// TIA Portal project "S7-1500 için Kod Çözücü(DECO) Komutu" (V18)

(* hardware
DEVICE "S7-1500/ET200MP station_1"  S7-1500 station
   slot 0: "Rail_0"  Rack  6ES7 590-1***0-0AA0
   slot 1: "PLC_1"  CPU 1512C-1 PN  6ES7 512-1CK00-0AB0  V2.8
      slot 3: "CPU display_1"  6ES7591-1AA00-0AA0
      slot 32768: "PROFINET interface_1"  X1
         slot 32769: "Port_1"  X1 P1
         slot 32770: "Port_2"  X1 P2
      slot 34817: "Virtual CP interface port_1"  Virtual CP interface port  Virtual CP interface port
*)

// ===== PLC "PLC_1"  CPU 1512C-1 PN =====

VAR_GLOBAL   // PLC tag table "Default tag table"
   "Tag_1" AT %I0.0 : Bool;
   "Tag_2" AT %MW10 : Int;
   "Tag_3" AT %Q0.0 : Bool;
   "Tag_4" AT %I0.1 : Bool;
   "Tag_5" AT %Q0.1 : Bool;
   "Tag_6" AT %MW11 : Int;
   "Tag_7" AT %MW12 : Int;
   "Tag_8" AT %MW13 : Int;
   "Tag_9" AT %MW14 : Int;
   "Tag_10" AT %I0.2 : Bool;
   "Tag_11" AT %I0.3 : Bool;
END_VAR

ORGANIZATION_BLOCK "Main"   // OB1, LAD, ProgramCycle
TITLE = "Main Program Sweep (Cycle)"
{ S7_Optimized_Access := 'TRUE' }
VERSION : 0.1
   VAR_INPUT
      Initial_Call : Bool;   // Initial call of this OB
      Remanence : Bool;   // =True, if remanent data are available
   END_VAR
BEGIN

REGION Network 1: MW10'a 5 değerini verdik.
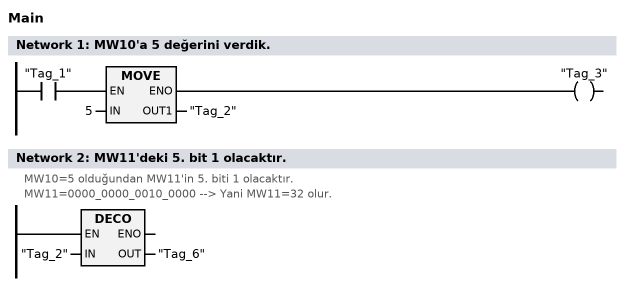
   RUNG wire#powerrail
      Contact( "Tag_1" )
      Move(in := 5, out1 => "Tag_2")
      Coil( "Tag_3" )
   END_RUNG
   // the same network as SCL:
   IF "Tag_1" THEN "Tag_2" := 5; END_IF;
   "Tag_3" := "Tag_1";
END_REGION

REGION Network 2: MW11'deki 5. bit 1 olacaktır.
   // MW10=5 olduğundan MW11'in 5. biti 1 olacaktır.
   // MW11=0000_0000_0010_0000 --> Yani MW11=32 olur.
   "Tag_6" := DECO(IN := "Tag_2");
END_REGION
END_ORGANIZATION_BLOCK